// TIA Portal project "teo1" (V15.1)

(* hardware
DEVICE "S7-1200 station_1"  S7-1200 Station
   slot 0: "Rack_0"  S7-1200 Rack  Rack  V1.0
   slot 1: "PLC_1"  CPU 1212FC DC/DC/RLY  6ES7 212-1HF40-0XB0  V4.2
*)

// ===== PLC "PLC_1"  CPU 1212FC DC/DC/RLY =====

VAR_GLOBAL   // PLC tag table "Tabla de variables estándar"
   "S1" AT %I0.0 : Bool;   // Sensor derecha
   "S2" AT %I0.1 : Bool;   // Sensor izquierda
   "S3" AT %I0.2 : Bool;   // Sensor vehiculo
   "M" AT %I0.3 : Bool;   // Marcha
   "P" AT %I0.4 : Bool;   // Paro
   "MP1" AT %Q0.0 : Bool;   // Motor Derecha -> Izquierda
   "MP2" AT %Q0.1 : Bool;   // Motor Izquierda -> Derecha
   "MV" AT %Q0.2 : Bool;   // Motor Ventilador
   "MC" AT %Q0.3 : Bool;   // Motor Cepillos
   "XV" AT %Q0.4 : Bool;   // Liquido
   "MARCA1" AT %M0.0 : Bool;   // Modo Marcha
   "MARCA2" AT %M0.1 : Bool;   // Modo lavado
   "MARCA3" AT %M0.2 : Bool;   // Modo vuelta lavado
   "MARCA4" AT %M0.3 : Bool;   // Modo ida secado
   "MARCA5" AT %M0.4 : Bool;   // Modo vuelta secado
   "MARCA6" AT %M0.5 : Bool;   // Modo emergencia
END_VAR

DATA_BLOCK "Main_Safety_RTG1_DB"   // DB1, F_DB
{ S7_Optimized_Access := 'TRUE' }
NAME : FUSI
VERSION : 0.1
// stored: InstanceOfName Main_Safety_RTG1
"Main_Safety_RTG1"
BEGIN
END_DATA_BLOCK

FUNCTION_BLOCK "Main_Safety_RTG1"   // FB1, F_FBD
{ S7_Optimized_Access := 'TRUE' }
VERSION : 0.1
BEGIN
END_FUNCTION_BLOCK

ORGANIZATION_BLOCK "Main"   // OB1, LAD, ProgramCycle
TITLE = "Main Program Sweep (Cycle)"
{ S7_Optimized_Access := 'TRUE' }
VERSION : 0.1
   VAR_INPUT
      Initial_Call : Bool;   // Initial call of this OB
      Remanence : Bool;   // =True, if remanent data are available
   END_VAR
BEGIN

REGION Network 1: Reposo a Activo - Inicio del proceso.
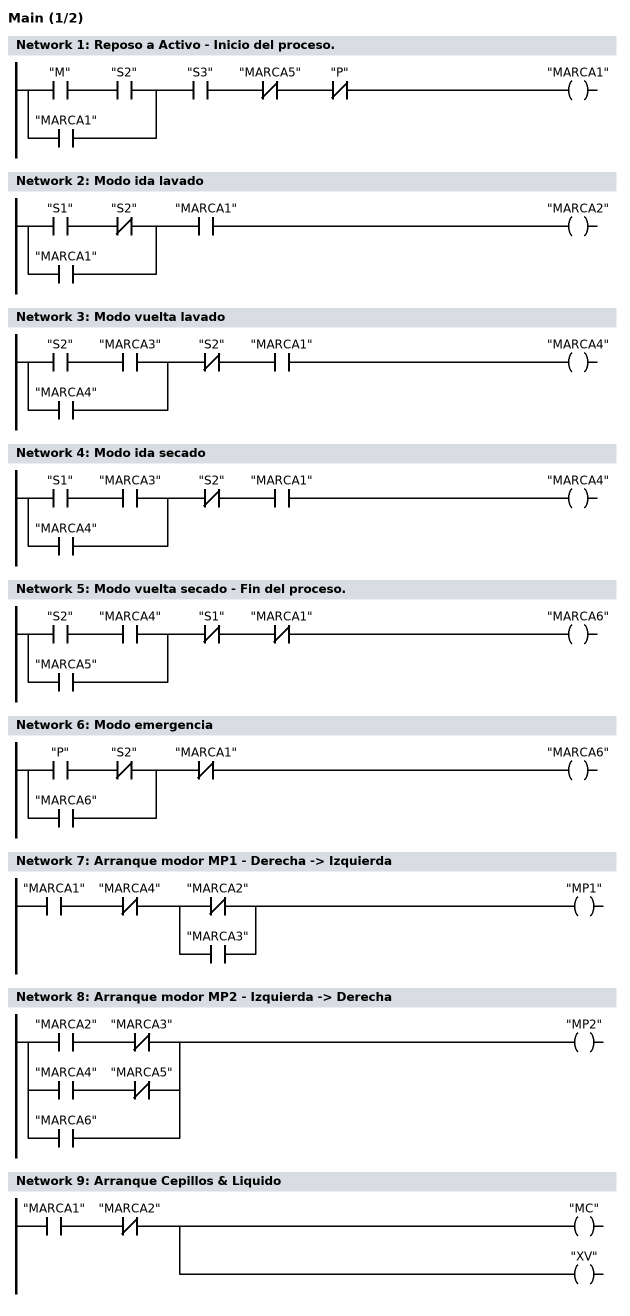
   RUNG wire#powerrail
      Contact( "M" )
      Contact( "S2" )
      wire#w1
      Contact( "S3" )
      I_Contact( "MARCA5" )
      I_Contact( "P" )
      Coil( "MARCA1" )
   END_RUNG
   RUNG wire#powerrail
      Contact( "MARCA1" )
   END_RUNG wire#w1
   // the same network as SCL:
   "MARCA1" := (("M" AND "S2") OR "MARCA1") AND "S3" AND NOT "MARCA5" AND NOT "P";
END_REGION

REGION Network 2: Modo ida lavado
   RUNG wire#powerrail
      Contact( "S1" )
      I_Contact( "S2" )
      wire#w1
      Contact( "MARCA1" )
      Coil( "MARCA2" )
   END_RUNG
   RUNG wire#powerrail
      Contact( "MARCA1" )
   END_RUNG wire#w1
   // the same network as SCL:
   "MARCA2" := (("S1" AND NOT "S2") OR "MARCA1") AND "MARCA1";
END_REGION

REGION Network 3: Modo vuelta lavado
   RUNG wire#powerrail
      Contact( "S2" )
      Contact( "MARCA3" )
      wire#w1
      I_Contact( "S2" )
      Contact( "MARCA1" )
      Coil( "MARCA4" )
   END_RUNG
   RUNG wire#powerrail
      Contact( "MARCA4" )
   END_RUNG wire#w1
   // the same network as SCL:
   "MARCA4" := (("S2" AND "MARCA3") OR "MARCA4") AND NOT "S2" AND "MARCA1";
END_REGION

REGION Network 4: Modo ida secado
   RUNG wire#powerrail
      Contact( "S1" )
      Contact( "MARCA3" )
      wire#w1
      I_Contact( "S2" )
      Contact( "MARCA1" )
      Coil( "MARCA4" )
   END_RUNG
   RUNG wire#powerrail
      Contact( "MARCA4" )
   END_RUNG wire#w1
   // the same network as SCL:
   "MARCA4" := (("S1" AND "MARCA3") OR "MARCA4") AND NOT "S2" AND "MARCA1";
END_REGION

REGION Network 5: Modo vuelta secado - Fin del proceso.
   RUNG wire#powerrail
      Contact( "S2" )
      Contact( "MARCA4" )
      wire#w1
      I_Contact( "S1" )
      I_Contact( "MARCA1" )
      Coil( "MARCA6" )
   END_RUNG
   RUNG wire#powerrail
      Contact( "MARCA5" )
   END_RUNG wire#w1
   // the same network as SCL:
   "MARCA6" := (("S2" AND "MARCA4") OR "MARCA5") AND NOT "S1" AND NOT "MARCA1";
END_REGION

REGION Network 6: Modo emergencia
   RUNG wire#powerrail
      Contact( "P" )
      I_Contact( "S2" )
      wire#w1
      I_Contact( "MARCA1" )
      Coil( "MARCA6" )
   END_RUNG
   RUNG wire#powerrail
      Contact( "MARCA6" )
   END_RUNG wire#w1
   // the same network as SCL:
   "MARCA6" := (("P" AND NOT "S2") OR "MARCA6") AND NOT "MARCA1";
END_REGION

REGION Network 7: Arranque modor MP1 - Derecha -> Izquierda
   RUNG wire#powerrail
      Contact( "MARCA1" )
      I_Contact( "MARCA4" )
      wire#w1
      I_Contact( "MARCA2" )
      wire#w2
      Coil( "MP1" )
   END_RUNG
   RUNG wire#w1
      Contact( "MARCA3" )
   END_RUNG wire#w2
   // the same network as SCL:
   "MP1" := "MARCA1" AND NOT "MARCA4" AND (NOT "MARCA2" OR "MARCA3");
END_REGION

REGION Network 8: Arranque modor MP2 - Izquierda -> Derecha
   RUNG wire#powerrail
      Contact( "MARCA2" )
      I_Contact( "MARCA3" )
      wire#w1
      Coil( "MP2" )
   END_RUNG
   RUNG wire#powerrail
      Contact( "MARCA4" )
      I_Contact( "MARCA5" )
   END_RUNG wire#w1
   RUNG wire#powerrail
      Contact( "MARCA6" )
   END_RUNG wire#w1
   // the same network as SCL:
   "MP2" := ("MARCA2" AND NOT "MARCA3") OR ("MARCA4" AND NOT "MARCA5") OR "MARCA6";
END_REGION

REGION Network 9: Arranque Cepillos & Liquido
   RUNG wire#powerrail
      Contact( "MARCA1" )
      I_Contact( "MARCA2" )
      wire#w1
      Coil( "MC" )
   END_RUNG
   RUNG wire#w1
      Coil( "XV" )
   END_RUNG
   // the same network as SCL:
   "MC" := "MARCA1" AND NOT "MARCA2";
   "XV" := "MC";
END_REGION

REGION Network 10: Arranque Ventilador
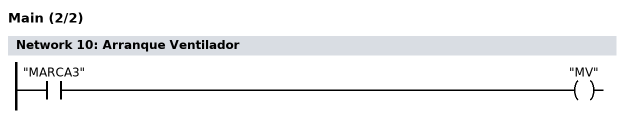
   RUNG wire#powerrail
      Contact( "MARCA3" )
      Coil( "MV" )
   END_RUNG
   // the same network as SCL:
   "MV" := "MARCA3";
END_REGION
END_ORGANIZATION_BLOCK